// TwinCAT 3 PLC project PLC1
// ProgramVersion: 3.1.4026.21
// libraries:
//   Tc2_Standard, * (Beckhoff Automation GmbH)
//   Tc2_System, * (Beckhoff Automation GmbH)
//   Tc3_Module, * (Beckhoff Automation GmbH)
// project tree:
//   DUTs/ Jog_FxA_Type.TcDUT, Jog_FxB_Type.TcDUT (not stored), LaserJog.TcDUT, LaserVar.TcDUT (not stored), Message_Type.TcDUT, MyCustomType.TcDUT (not stored), SideClampVar.TcDUT (not stored), XYZ_Point.TcDUT
//   GVLs/ GVL.TcGVL (not stored), GVL_Main.TcGVL, Hmi_web.TcGVL
//   / PlcTask.TcTTO (not stored)
//   POUs/ MAIN.TcPOU (not stored)
// real-time tasks:
//   TASK PlcTask: cycle T#10ms, priority 20, ADS port 350

// ---- DUTs/Jog_FxA_Type.TcDUT
TYPE Jog_FxA_Type :
STRUCT
	
 H_Open:  BOOL;
 H_Open_S:  BOOL;
 H_Close:  BOOL;
 H_Close_S:  BOOL;

 H_Hold:  BOOL;
 H_Hold_S:  BOOL;

 V_Open:  BOOL;
 V_Open_S: BOOL;
 V_Close: BOOL;
 V_Close_S: BOOL;
  P : BOOL;
 P_S : BOOL;
 N : BOOL;
 N_S : BOOL;
 P_Fast : BOOL;
 P_Fast_S : BOOL;
 N_Fast : BOOL;
 N_Fast_S : BOOL;
END_STRUCT
END_TYPE

// ---- DUTs/LaserJog.TcDUT
TYPE LaserJog :
STRUCT
	 X_P: BOOL;
     X_N: BOOL;
     X_H: BOOL;
	 
	 
	 X_P_S: BOOL;
     X_N_S: BOOL;
     X_H_S: BOOL;
	 
     Y_P: BOOL;
     Y_N: BOOL;
     Y_H: BOOL;
	 
	 
     Y_P_S: BOOL;
     Y_N_S: BOOL;
     Y_H_S: BOOL;
	 
     Z_P: BOOL;
     Z_N: BOOL;
     Z_H: BOOL;
	 
     Z_P_S: BOOL;
     Z_N_S: BOOL;
     Z_H_S: BOOL;
     Laser_Preview:BOOL;
     Laser_Preview_Select: INT;
     Laser_Blow: BOOL;
     Laser_Cover: BOOL;
	 
	 Pos:XYZ_Point;

END_STRUCT
END_TYPE

// ---- DUTs/Message_Type.TcDUT
TYPE Message_Type :
STRUCT
	  sv_iActAlarmCount: INT; ////錯誤數量
      sv_Alarms: STRING; //警告(陣列)
      sv_bMessageResetAll: BOOL; //重置所有警報 boolean
      sv_bMessageQuitAll: BOOL; //確認所有警報 boolean
      sv_bMessageResetSelected: BOOL; //重置選定的警報 boolean
      sv_bMessageQuitSelected: BOOL; //確認選定的警報 boolean
      sv_iSelectedAlarmIndex: INT; //清除選定的警報 int
      sv_bMessageUpdateAlarms: BOOL; //更新警報列表的觸發器 boolean
END_STRUCT
END_TYPE

// ---- DUTs/XYZ_Point.TcDUT
TYPE XYZ_Point :
STRUCT
	X:LREAL;
	Y:LREAL;
	Z:LREAL;
END_STRUCT
END_TYPE

// ---- GVLs/GVL_Main.TcGVL
{attribute 'qualified_only'}
VAR_GLOBAL
    g_bStart     : BOOL := FALSE;
    g_iCounter   : INT := 0;
    g_fSpeed     : REAL := 1.5;
    testBoolean     : BOOL := FALSE;
	
 g_machineStatus : MyCustomType := (
        isActive := FALSE,
        speed    := 0.0,
        counter  := 0
    );
	

LaserVars1:LaserVar := (
sv_bPLCHandShaking:= FALSE,
sv_bIPCHandShaking:= FALSE
    );
	LaserVars2:LaserVar := (
sv_bPLCHandShaking:= FALSE,
sv_bIPCHandShaking:= FALSE
    );
	LaserVars3:LaserVar := (
sv_bPLCHandShaking:= FALSE,
sv_bIPCHandShaking:= FALSE
    );
	LaserVars4:LaserVar := (
sv_bPLCHandShaking:= FALSE,
sv_bIPCHandShaking:= FALSE
    );

	
SideClampVars1:SideClampVar := (
sv_bButtonFwd:= FALSE,
sv_bButtonBwd:= FALSE);
	
SideClampVars2:SideClampVar := (
sv_bButtonFwd:= FALSE,
sv_bButtonBwd:= FALSE
 );
	
	

	
	
	
	
	
	
	
	
END_VAR

// ---- GVLs/Hmi_web.TcGVL
{attribute 'qualified_only'}
VAR_GLOBAL
	// 點動速度
    Jog_Speed: INT;
	
 Oil_Pump:BOOL;
Jog_FxA:Jog_FxA_Type:= (
      H_Open:= FALSE,
      H_Open_S:= FALSE,
      H_Close:= FALSE,
      H_Close_S:= FALSE,

      H_Hold:= FALSE,
      H_Hold_S:= FALSE,

      V_Open:= FALSE,
      V_Open_S:= FALSE,
      V_Close:= FALSE,
      V_Close_S:= FALSE,
   
     P:= FALSE,
      P_S:= FALSE,
      N:= FALSE,
      N_S:= FALSE,
      P_Fast:= FALSE,
      P_Fast_S:= FALSE,
      N_Fast:= FALSE,
      N_Fast_S:= FALSE
    );
 
 
Jog_FxB : Jog_FxB_Type := (
       H_Open:= FALSE,
      H_Open_S:= FALSE,
      H_Close:= FALSE,
      H_Close_S:= FALSE,

      H_Hold:= FALSE,
      H_Hold_S:= FALSE,

      V_Open:= FALSE,
      V_Open_S:= FALSE,
      V_Close:= FALSE,
      V_Close_S:= FALSE

    
);


 

//右軸
Jog_Ga: LaserJog:=( 
     X_P:= FALSE,
     X_N:= FALSE,
     X_H:= FALSE,
     Y_P:= FALSE,
     Y_N:= FALSE,
     Y_H:= FALSE,
     Z_P:= FALSE,
     Z_N:= FALSE,
     Z_H:= FALSE,
     Laser_Preview:=FALSE,
     Laser_Preview_Select:= 1,
     Laser_Blow:= FALSE,
     Laser_Cover:= FALSE);
//上軸
    Jog_Gb: LaserJog:=( 
     X_P:= FALSE,
     X_N:= FALSE,
     X_H:= FALSE,
     Y_P:= FALSE,
     Y_N:= FALSE,
     Y_H:= FALSE,
     Z_P:= FALSE,
     Z_N:= FALSE,
     Z_H:= FALSE,
     Laser_Preview:=FALSE,
     Laser_Preview_Select:= 1,
     Laser_Blow:= FALSE,
     Laser_Cover:= FALSE);
//左軸
    Jog_Gc: LaserJog:=( 
     X_P:= FALSE,
     X_N:= FALSE,
     X_H:= FALSE,
     Y_P:= FALSE,
     Y_N:= FALSE,
     Y_H:= FALSE,
     Z_P:= FALSE,
     Z_N:= FALSE,
     Z_H:= FALSE,
     Laser_Preview:=FALSE,
     Laser_Preview_Select:= 1,
     Laser_Blow:= FALSE,
     Laser_Cover:= FALSE);
//下軸
    Jog_Gd: LaserJog:=( 
     X_P:= FALSE,
     X_N:= FALSE,
     X_H:= FALSE,
     Y_P:= FALSE,
     Y_N:= FALSE,
     Y_H:= FALSE,
     Z_P:= FALSE,
     Z_N:= FALSE,
     Z_H:= FALSE,
     Laser_Preview:=FALSE,
     Laser_Preview_Select:= 1,
     Laser_Blow:= FALSE,
     Laser_Cover:= FALSE);

	 // 左側-XYZ座標
	 Ga_Pos:XYZ_Point:=(
		X:=0,
		Y:=0,
		Z:=0
		);
	 // 上方-XYZ座標
	Gb_Pos:XYZ_Point:=(
		X:=0,
		Y:=0,
		Z:=0
		);
	 // 右側-XYZ座標
	Gc_Pos:XYZ_Point:=(
		X:=0,
		Y:=0,
		Z:=0
		);
	 // 下方-XYZ座標
	Gd_Pos:XYZ_Point:=(
		X:=0,
		Y:=0,
		Z:=0
		);
	 
	 
	 
	 
	 

 	//*自動加工 */
    Auto_Start:  BOOL;
    //插單*/
    Auto_OneCycle_Start:  BOOL;
 	// 自動流程 加工單
	Auto_ProjectWorkOrder_uuid: STRING;
	// 排版專案 
    Start_WorkOrder_UUID: STRING;
	
	// Top 右 加工data_uuid
    Process_Data_UUID_A: STRING;
	// Top 右 雷標動作啟動 
    Process_Data_UUID_A_Start: BOOL;
	// Front 上 加工data_uuid
    Process_Data_UUID_B: STRING;
	// Front 上 雷標動作啟動 
    Process_Data_UUID_B_Start: BOOL;
	// Bottom 左 加工data_uuid
    Process_Data_UUID_C: STRING;
	// Bottom 左 雷標動作啟動 
    Process_Data_UUID_C_Start: BOOL;
	// Behind 下 加工data_uuid 
    Process_Data_UUID_D: STRING;
	// Behind 下 雷標動作啟動 
    Process_Data_UUID_D_Start: BOOL;
	

	// 預覽模式
	Preview_Enable:BOOL;
	// 原點復歸
	Auto_homming:BOOL;
 
 

    //動力滾輪
    Roller_Fwd:  BOOL;
    Roller_Fwd_S:  BOOL;
    //動力滾輪反轉
    Roller_Rev:  BOOL;
    Roller_Rev_S:  BOOL;

    //滾輪上浮
    Roller_Up:  BOOL;
    Roller_Up_S:  BOOL;
    //滾輪下降
    Roller_Down:  BOOL;
    Roller_Down_S:  BOOL;

    //入口料架-出口料架(0/1)*/
    Site_Select:  INT;
    //料架速率(0/1)*/
    Speed_Select:  INT;

    // 指定橫移->用二進位儲存 */
    Module_Select:  INT;

    //料架動作-台車前進*/
    Car_Rev:  BOOL;
    Car_Rev_S:  BOOL;
    //料架動作-台車後退
    Car_Fwd:  BOOL;
    Car_Fwd_S:  BOOL;
    //料架動作-台車上升
    Car_Up: BOOL;
    Car_Up_S:  BOOL;
    //料架動作-台車中間
    Car_Midd:  BOOL;
    Car_Midd_S:  BOOL;

    //料架動作-台車下降
    Car_Down:  BOOL;
    Car_Down_S:  BOOL;

    //料架動作-靠邊
    Pull_over_Push: BOOL;
    Pull_over_Push_S: BOOL;

    //料架動作-頂料柱上升
    StopPin_Up: BOOL;
    StopPin_Up_S:  BOOL;

    //料架動作-頂料柱下降
    StopPin_Down: BOOL;
    StopPin_Down_S: BOOL;

MessageVar1:Message_Type:=( 
      sv_iActAlarmCount:=0, //錯誤數量
      sv_Alarms:= '', //警告(陣列)
      sv_bMessageResetAll:= FALSE, //重置所有警報 boolean
      sv_bMessageQuitAll:= FALSE, //確認所有警報 boolean
      sv_bMessageResetSelected:= FALSE, //重置選定的警報 boolean
      sv_bMessageQuitSelected:= FALSE, //確認選定的警報 boolean
      sv_iSelectedAlarmIndex:= 0, //清除選定的警報 int
      sv_bMessageUpdateAlarms:= FALSE //更新警報列表的觸發器 boolean
    );



END_VAR
